FUNCTION_BLOCK fbCylinder EXTENDS fbComponent IMPLEMENTS ICylinder
VAR_INPUT
	(*~
		<docu>
			<summary>
				Home position sensor.
			</summary>	
		</docu>
	~*)
	{attribute wpf [Container(Layout.UniformGrid)]}
	{attribute wpf [Group(Layout.GroupBox, "Inputs")]}	
	{attribute addProperty Name "Home position sensor"}
	inAtHomePos : BOOL;
	(*~
		<docu>
			<summary>
				Working position sensor.
			</summary>	
		</docu>
	~*) 
	{attribute addProperty Name "Work position sensor"}
	inAtWorkPos : BOOL; 
END_VAR
VAR_OUTPUT
	(*~
		<docu>
			<summary>
				Move to working home position signal.
			</summary>	
		</docu>
	~*)
	{attribute wpf [Container(Layout.UniformGrid)]}
	{attribute wpf [Group(Layout.GroupBox, "Outputs")]}	
	{attribute addProperty Name "Move to home position actuator"}
	outToHomePos : BOOL;
	(*~
		<docu>
			<summary>
				Move to working posistion signal.
			</summary>	
		</docu>
	~*)
	{attribute addProperty Name "Move to work position actuator"}
	outToWorkPos : BOOL;
END_VAR

VAR	
	{attribute wpf [Container(Layout.UniformGrid)]}
	{attribute addProperty Name "Request move to Home position"}	
	_moveHomeTask : fbTask(THIS^);
	{attribute addProperty Name "Request move to Work position"}
	_moveWorkTask : fbTask(THIS^);
	{attribute addProperty Name "Request Stop"}
	_stopTask : fbTask(THIS^);
END_VAR

IF(_moveHomeTask.Execute(1)) THEN
	outToHomePos := TRUE;
	outToWorkPos := FALSE; 		
	_moveHomeTask.DoneWhen(inAtHomePos);			
END_IF

IF(_moveWorkTask.Execute(2)) THEN
	outToWorkPos := TRUE; 
	outToHomePos := FALSE;
	_moveWorkTask.DoneWhen(inAtWorkPos);
END_IF;	 

IF(_stopTask.Execute(0)) THEN	
	outToWorkPos := FALSE; 
	outToHomePos := FALSE;
	_moveWorkTask.Reset();
	_moveHomeTask.Reset();
	_stopTask.Reset();
	_stopTask.DoneWhen(TRUE);	
END_IF

{attribute 'TcRpcEnable'}
METHOD INTERNAL _MoveToHomeTest : BOOL
_MoveToHomeTest := MoveToHome().Done;
END_METHOD

{attribute 'TcRpcEnable'}
METHOD INTERNAL _MoveToWorkTest : BOOL
_MoveToWorkTest := MoveToWork().Done;
END_METHOD

{attribute 'TcRpcEnable'}
METHOD INTERNAL _StopTest : BOOL
_StopTest := Stop().Done;
END_METHOD

PROPERTY AtHome : bool
GET
AtHome := inAtHomePos;
END_GET
END_PROPERTY

PROPERTY AtWork : bool
GET
AtWork := inAtWorkPos;
END_GET
END_PROPERTY

METHOD PROTECTED  ManualControl
END_METHOD

(*~
	<docu>
		<summary>
			Moves the piston into home position.
		</summary>
		<returns>True when home position sensor is reached.</returns>
	</docu>
~*)
METHOD MoveToHome : ITaskStatus
THIS^._moveHomeTask.Invoke();
MoveToHome := THIS^._moveHomeTask;
END_METHOD

(*~
	<docu>
		<summary>
			Moves the piston into working position.
		</summary>
		<returns>True when working position sensor is reached.</returns>
	</docu>
~*)
METHOD MoveToWork : ITaskStatus
THIS^._moveWorkTask.Invoke();
MoveToWork := THIS^._moveWorkTask;
END_METHOD

METHOD Stop : REFERENCE TO fbTask
_stopTask.Invoke();
Stop REF= _stopTask;
END_METHOD

END_FUNCTION_BLOCK

(* stored: Version 1.1.0.1, ProductVersion 3.1.4024.5
   POU fbCylinder: Id {fe4e2550-76ec-4019-82bb-e68b2cbe4d49}, SpecialFunc None
   Folder _tests: Id {2cbd4d6b-2a4a-49b8-b437-ed7c5a45b843}
   Method _MoveToHomeTest: Id {9ef39d14-16a3-4bc8-b330-33d879f1f7f9}
   Method _MoveToWorkTest: Id {7ebcdca4-683e-48c8-8052-33f48bfaaa19}
   Method _StopTest: Id {28dff165-f4ab-484d-9c26-93aee0eaf841}
   Property AtHome: Id {d06903a0-9230-4f9a-9ffc-ed1726b8d4b9}
   Get Get: Id {2309dcb2-6c63-44cf-85e0-e6e2754836eb}
   Property AtWork: Id {c484892b-8ab6-4a33-a377-7a200a12d81a}
   Get Get: Id {b963dd74-98d0-4492-a086-b714bde49f51}
   Method ManualControl: Id {94b70f4e-af12-4cab-8a9f-9a3da438ebd4}
   Method MoveToHome: Id {40560f4f-3063-47a8-8b62-1f2968f73b89}
   Method MoveToWork: Id {d11735f5-ce5f-4a7f-8109-144749721e33}
   Method Stop: Id {9e32cbb8-ba72-4463-bbd6-9f7b9b0e82cd} *)
